screen "05_Receipt" 800x480, template "MainTemplate"
   TextField "Text field_1" at 258,159 size 300x124; Text 'KAYDEDİLDİ'
      Visibility <- "Receipt_bShowMessage"
   TextField "Template_Text field_1" at 45,17 size 109x22; Text 'Model Seçimi:'
   SymbolicIOField "Template_Symbolic I/O field_1" at 270,13 size 524x32; TextOn '1'; TextOff '0'; TextList "textListReceipt"
      ProcessValue <- "ModelId"
   Button "btnSave" at 619,337 size 167x58; TextOff 'KAYDET'
      on Release: SetBit("Receipt_btnSave")
   TextField "Template_Text field_4" at 45,139 size 124x22; Text 'Model Boyu (C):'
   TextField "Template_Text field_2" at 46,57 size 83x22; Text 'Model Adı:'
   IOField "I/O field_1" at 274,53 size 524x32; FormatPattern ??????????????????????????????????????????????????
      ProcessValue <- "ModelName"
   IOField "I/O field_2" at 273,134 size 256x32; FormatPattern s9999999.99; Unit  mm
      ProcessValue <- "Receipt_CurrentModel_Boy_C"
   TextField "Template_Text field_5" at 46,181 size 111x22; Text 'Model Eni (D):'
   IOField "I/O field_3" at 274,175 size 256x32; FormatPattern s9999999.99; Unit  mm
      ProcessValue <- "Receipt_CurrentModel_En_D"
   TextField "Template_Text field_3" at 45,98 size 99x22; Text 'Model Sınıfı:'
   SymbolicIOField "Template_Symbolic I/O field_2" at 275,94 size 68x32; TextOn '1'; TextOff '0'; TextList "classList"
      ProcessValue <- "Receipt_CurrentModel_Class"
   IOField "I/O field_4" at 275,290 size 185x32; FormatPattern 99999.99; Unit  mm
      ProcessValue <- "HMI_Data_ServoData_txtGerdirmeMes"
   TextField "Template_Text field_6" at 46,294 size 151x22; Text 'Gerdirme Mesafesi:'
   TextField "Template_Text field_7" at 45,252 size 154x23; Text 'Kenetleme Süresi:'
   IOField "Template_I/O field_1" at 275,248 size 184x32; FormatPattern 9999999999; Unit  sn
      ProcessValue <- "HMI_Data_KenetlemeSuresi"

screen "06_Alarm" 800x480, template "MainTemplate"
   AlarmView "Alarm view_1" at 2,1 size 796x415

screen "Screen_1" 800x480
   TextField "Text field_4" at 293,58 size 227x20; Text 'SERVO OTOMATİK KONTROL'
   IOField "I/O field_4" at 304,101 size 202x39; FormatPattern 999.9; Unit  %
      ProcessValue <- "HMI_Data_ServoData_txtVelocity"
   TextField "Text field_6" at 74,110 size 134x20; Text 'OTOMATİK MOD HIZ:'
   Button "btnIncJogSpeedXaxis_1" at 224,102 size 74x37; TextOff '-'
      on Release: function_b9b71300("HMI_Data_ServoData_txtVelocity", 5)
   Button "Button_1" at 512,102 size 75x37; TextOff '+'
      on Release: function_dd21b452("HMI_Data_ServoData_txtVelocity", 5)
*)